FUNCTION_BLOCK fValve

VAR_IN_OUT
	valv:dutValve;
END_VAR

VAR
	a: INT;
	tonFailFCOp: Ton;
	tonFailFCCl: Ton;
	bFailFCop:BOOL;	(*Fail FC*)
	bFailFCcl:BOOL;	(*Fail FC*)
	test: BOOL;
	tToFail: TIME := T#5S;
END_VAR

a:=a+1;

valv.xFailFC:=FALSE;
valv.xFailFCc:=FALSE;
valv.xFailFCo:=FALSE;
		
(*=========================================================================================================*)
(*Salida  BECHOFF DO*)
				
(*FC valve open*)
tonFailFCOp(IN:= (valv.xOpen)AND NOT(valv.xFailFCo) , PT:=tToFail );
valv.xFailFCo:= tonFailFCOp.Q;

(*FC valve close*)
tonFailFCCl(IN:= NOT(valv.xOpen)AND NOT(valv.xFailFCc) , PT:=tToFail  );
valv.xFailFCc:= tonFailFCCl.Q;

(*FC Valve*)		
valv.xFailFC:= valv.xFailFCo OR valv.xFailFCc;

(*=========================================================================================================*)

END_FUNCTION_BLOCK

(* stored: Version 1.1.0.1, ProductVersion 3.1.4024.12
   POU fValve: Id {de76ec87-4c68-4a40-bf4d-7a95fb3a12ac}, SpecialFunc None *)
